# EPICS substitutions: apps/mpodLvApp/Db/fthodlv.substitutions
file "db/mpod8008l.db" {
    pattern {HOST,CH,SCAN,PORT,DETALIAS}
{"129.57.86.109","100","2 second","B_HW_LVFTAG_Sl1_Ch0","B_DET_FTH_LV_Sl1_Ch0"}
{"129.57.86.109","101","2 second","B_HW_LVFTAG_Sl1_Ch1","B_DET_FTH_LV_Sl1_Ch1"}
{"129.57.86.109","102","2 second","B_HW_LVFTAG_Sl1_Ch2","B_DET_FTH_LV_Sl1_Ch2"}
{"129.57.86.109","103","2 second","B_HW_LVFTAG_Sl1_Ch3","B_DET_FTH_LV_Sl1_Ch3"}
{"129.57.86.109","104","2 second","B_HW_LVFTAG_Sl1_Ch4","B_DET_FTH_LV_Sl1_Ch4"}
{"129.57.86.109","105","2 second","B_HW_LVFTAG_Sl1_Ch5","B_DET_FTH_LV_Sl1_Ch5"}
{"129.57.86.109","106","2 second","B_HW_LVFTAG_Sl1_Ch6","B_DET_FTH_LV_Sl1_Ch6"}
}
